// TIA Portal project "tram4_duy" (V16)

(* hardware
DEVICE "S7-1200 station_1"  S7-1200 Station
   slot 0: "Rack_0"  S7-1200 Rack  Rack  V1.0
   slot 1: "PLC_1"  CPU 1214C AC/DC/Rly  6ES7 214-1BG40-0XB0  V4.2
*)

// ===== PLC "PLC_1"  CPU 1214C AC/DC/Rly =====

VAR_GLOBAL   // PLC tag table "Default tag table"
   "Tag_1" AT %I1.1 : Bool;
   "M1" AT %Q0.0 : Bool;
   "Tag_3" AT %I1.0 : Bool;
   "Tag_4" AT %Q0.1 : Bool;
   "M3" AT %Q0.6 : Bool;
   "quaynghich" AT %Q0.7 : Bool;
   "start" AT %I0.6 : Bool;
   "stop" AT %I1.5 : Bool;
   "Tag_7" AT %M0.1 : Bool;
   "Tag_5" AT %M0.0 : Bool;
   "Tag_6" AT %Q0.2 : Bool;
   "M2" AT %Q0.3 : Bool;
   "Tag_9" AT %Q0.4 : Bool;
   "Tag_10" AT %Q0.5 : Bool;
   "Tag_2" AT %M1.0 : Bool;
   "Tag_8" AT %M1.1 : Bool;
   "Tag_11" AT %M1.2 : Bool;
   "Tag_12" AT %M2.0 : Bool;
   "Tag_13" AT %M2.1 : Bool;
   "Tag_14" AT %M2.2 : Bool;
   "Tag_15" AT %Q1.0 : Bool;
   "Tag_16" AT %Q1.1 : Bool;
END_VAR

// folder: System blocks/Program resources

DATA_BLOCK "T1"   // DB1
{ S7_Optimized_Access := 'TRUE' }
AUTHOR : Simatic
FAMILY : IEC
NAME : IEC_TMR
VERSION : 1.0
// stored: InstanceOfName IEC_TIMER
"IEC_TIMER"
BEGIN
END_DATA_BLOCK

DATA_BLOCK "T2"   // DB2
{ S7_Optimized_Access := 'TRUE' }
AUTHOR : Simatic
FAMILY : IEC
NAME : IEC_TMR
VERSION : 1.0
// stored: InstanceOfName IEC_TIMER
"IEC_TIMER"
BEGIN
END_DATA_BLOCK

DATA_BLOCK "T3"   // DB3
{ S7_Optimized_Access := 'TRUE' }
AUTHOR : Simatic
FAMILY : IEC
NAME : IEC_TMR
VERSION : 1.0
// stored: InstanceOfName IEC_TIMER
"IEC_TIMER"
BEGIN
END_DATA_BLOCK

DATA_BLOCK "T4"   // DB4
{ S7_Optimized_Access := 'TRUE' }
AUTHOR : Simatic
FAMILY : IEC
NAME : IEC_TMR
VERSION : 1.0
// stored: InstanceOfName IEC_TIMER
"IEC_TIMER"
BEGIN
END_DATA_BLOCK

// folder: (top level)

ORGANIZATION_BLOCK "Main"   // OB1, LAD, ProgramCycle
TITLE = "Main Program Sweep (Cycle)"
{ S7_Optimized_Access := 'TRUE' }
VERSION : 0.1
   VAR_INPUT
      Initial_Call : Bool;   // Initial call of this OB
      Remanence : Bool;   // =True, if remanent data are available
   END_VAR
BEGIN

REGION Network 1
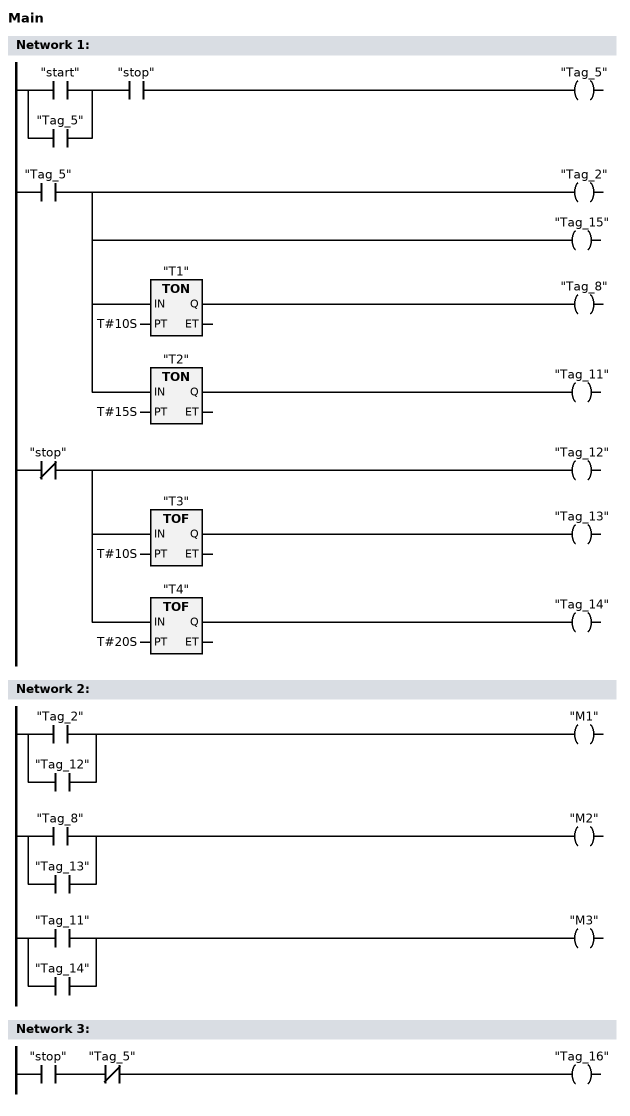
   "Tag_5" := ("start" OR "Tag_5") AND "stop";
   "Tag_2" := "Tag_5";
   "Tag_15" := "Tag_5";
   "T1".TON(IN := "Tag_5", PT := T#10S);
   "Tag_8" := "T1".Q;
   "T2".TON(IN := "Tag_5", PT := T#15S);
   "Tag_11" := "T2".Q;
   "Tag_12" := NOT "stop";
   "T3".TOF(IN := NOT "stop", PT := T#10S);
   "Tag_13" := "T3".Q;
   "T4".TOF(IN := NOT "stop", PT := T#20S);
   "Tag_14" := "T4".Q;
END_REGION

REGION Network 2
   RUNG wire#powerrail
      Contact( "Tag_2" )
      wire#w1
      Coil( "M1" )
   END_RUNG
   RUNG wire#powerrail
      Contact( "Tag_12" )
   END_RUNG wire#w1
   RUNG wire#powerrail
      Contact( "Tag_8" )
      wire#w2
      Coil( "M2" )
   END_RUNG
   RUNG wire#powerrail
      Contact( "Tag_13" )
   END_RUNG wire#w2
   RUNG wire#powerrail
      Contact( "Tag_11" )
      wire#w3
      Coil( "M3" )
   END_RUNG
   RUNG wire#powerrail
      Contact( "Tag_14" )
   END_RUNG wire#w3
   // the same network as SCL:
   "M1" := "Tag_2" OR "Tag_12";
   "M2" := "Tag_8" OR "Tag_13";
   "M3" := "Tag_11" OR "Tag_14";
END_REGION

REGION Network 3
   RUNG wire#powerrail
      Contact( "stop" )
      I_Contact( "Tag_5" )
      Coil( "Tag_16" )
   END_RUNG
   // the same network as SCL:
   "Tag_16" := "stop" AND NOT "Tag_5";
END_REGION
END_ORGANIZATION_BLOCK